{attribute 'hide_all_locals'}
FUNCTION_BLOCK AxesReset EXTENDS TaskBase
VAR_INPUT
END_VAR
VAR_OUTPUT
END_VAR
VAR
	resetMover : Tc2_MC2.MC_Reset;
	_Axis : REFERENCE TO Tc2_MC2.AXIS_REF;
	_ResetMover : BOOL;
END_VAR

{analysis -2}

METHOD Abort : BOOL
resetMover.Execute := FALSE;
_Busy := FALSE;
_ResetMover := FALSE;
Abort := TRUE;
State := 0;
END_METHOD

METHOD Cycle : HRESULT
VAR_INPUT
END_VAR
CASE State OF
	0:
		IF _ResetMover THEN
			Cycle := S_PENDING;
			_Done := FALSE;
			_Error := FALSE;
			_Busy := TRUE;
			resetMover.Execute := TRUE;
			IF resetMover.Busy THEN
				State := 10;
				_ResetMover := FALSE;
			END_IF
		END_IF
	
	10:
		IF NOT resetMover.Busy THEN
			IF resetMover.Done THEN
				_Done := TRUE;
			ELSIF resetMover.Error THEN
				_Error := TRUE;
			END_IF
			_Busy := FALSE;
			resetMover.Execute := FALSE;
			State := 0;
			Cycle := S_OK;
		END_IF
END_CASE

resetMover(Axis := _Axis);
END_METHOD

METHOD Execute : BOOL
VAR_INPUT
END_VAR
Execute := _ResetMover := true;
END_METHOD

METHOD FB_init : BOOL
VAR_INPUT
	bInitRetains : BOOL; // if TRUE, the retain variables are initialized (warm start / cold start)
	bInCopyCode : BOOL;  // if TRUE, the instance afterwards gets moved into the copy code (online change)
	axis : reference TO AXIS_REF;
END_VAR
_Axis REF= axis;
END_METHOD

END_FUNCTION_BLOCK

(* stored: Version 1.1.0.1, ProductVersion 3.1.4024.12
   POU AxesReset: Id {ea00788b-a7e2-4ddb-a987-8527d11bfcf5}, SpecialFunc None
   Method Abort: Id {175585a1-cdb8-4dd4-9630-03b10e9f2656}
   Method Cycle: Id {a2f61a2f-8d99-4872-967a-55fbf379e9cf}
   Method Execute: Id {3351ec6f-5e58-4cce-afac-76b6f35f5e04}
   Method FB_init: Id {9a079dc9-6267-424b-87ad-35fb5655339d} *)
